% RSLogix 500 project PROC1.RSS, saved by version 8.30.00.16 %
PROJECT "UNTITLED"    % processor: Bul.1763 MicroLogix 1100 Series B %

PROGRAM FILES
  LAD 2 "MAIN"  5 rungs
  LAD 3 "ALARMS"  1 rungs
  LAD 4 "DIGITAL IO"  9 rungs
  LAD 5 "CONTROLS"  1 rungs
  LAD 6 "ANALOG IO"  8 rungs

DATA FILES
  O0 OUTPUT  9 elements
  I1 INPUT  19 elements
  S2 STATUS  66 elements
  B3 BINARY  1 elements
  T4 TIMER  1 elements
  C5 COUNTER  1 elements
  R6 CONTROL  1 elements
  N7 INTEGER  1 elements
  F8 FLOAT  1 elements

LADDER 2 "MAIN"
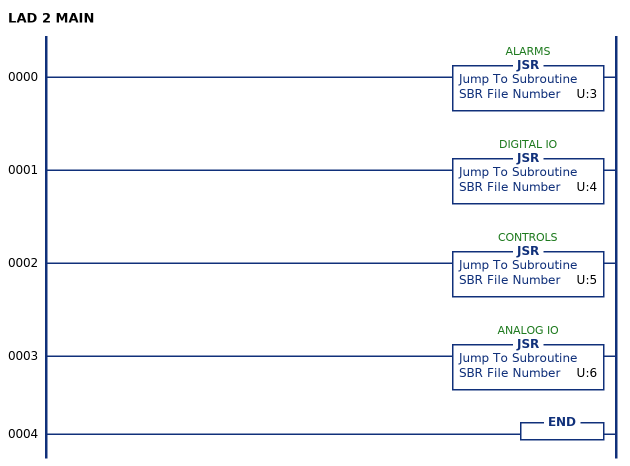
% Rung: 0 %  % edit flag set %
SOR JSR U:3 EOR
%   U:3  "ALARMS" %
% Rung: 1 %
SOR JSR U:4 EOR
%   U:4  "DIGITAL IO" %
% Rung: 2 %  % edit flag set %
SOR JSR U:5 EOR
%   U:5  "CONTROLS" %
% Rung: 3 %  % edit flag set %
SOR JSR U:6 EOR
%   U:6  "ANALOG IO" %
% Rung: 4 %
SOR END EOR

LADDER 4 "DIGITAL IO"
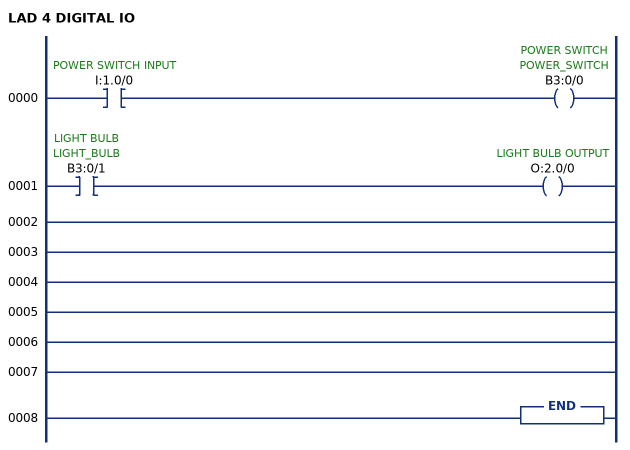
% Rung: 0 %  % edit flag set %
SOR XIC I:1.0/0 OTE B3:0/0 EOR
%   I:1.0/0  "POWER SWITCH INPUT" %
%   B3:0/0  POWER_SWITCH  "POWER SWITCH" %
% Rung: 1 %  % edit flag set %
SOR XIC B3:0/1 OTE O:2.0/0 EOR
%   B3:0/1  LIGHT_BULB  "LIGHT BULB" %
%   O:2.0/0  "LIGHT BULB OUTPUT" %
% Rung: 2 %  % edit flag set %
SOR EOR
% Rung: 3 %  % edit flag set %
SOR EOR
% Rung: 4 %  % edit flag set %
SOR EOR
% Rung: 5 %  % edit flag set %
SOR EOR
% Rung: 6 %  % edit flag set %
SOR EOR
% Rung: 7 %  % edit flag set %
SOR EOR
% Rung: 8 %
SOR END EOR

LADDER 6 "ANALOG IO"
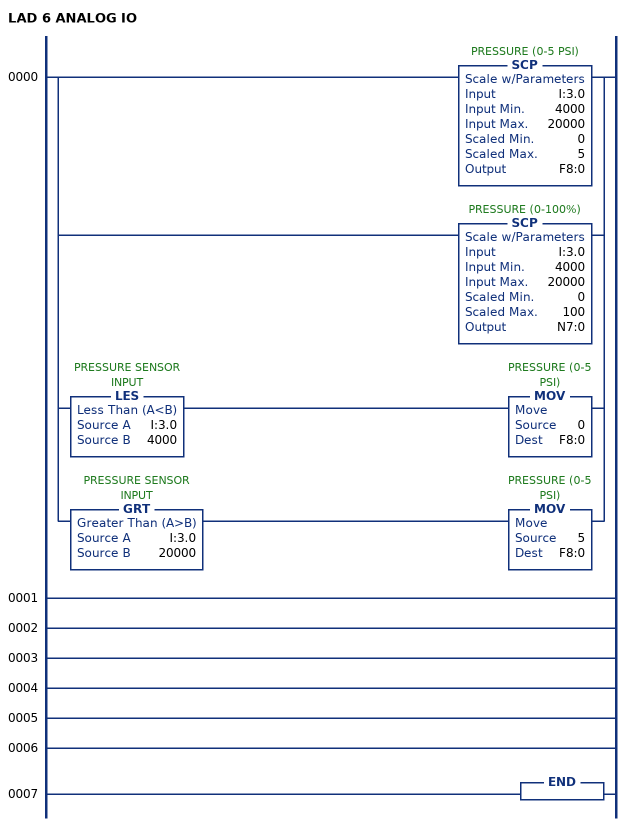
% Rung: 0 %  % edit flag set %
SOR BST SCP I:3.0 4000 20000 0 5 F8:0 NXB SCP I:3.0 4000 20000 0 100 N7:0 NXB LES I:3.0 4000 MOV 0 F8:0 NXB GRT I:3.0 20000 MOV 5 F8:0 BND EOR
%   I:3.0  "PRESSURE SENSOR INPUT" %
%   F8:0  "PRESSURE (0-5 PSI)" %
%   N7:0  "PRESSURE (0-100%)" %
% Rung: 1 %  % edit flag set %
SOR EOR
% Rung: 2 %  % edit flag set %
SOR EOR
% Rung: 3 %  % edit flag set %
SOR EOR
% Rung: 4 %  % edit flag set %
SOR EOR
% Rung: 5 %  % edit flag set %
SOR EOR
% Rung: 6 %  % edit flag set %
SOR EOR
% Rung: 7 %
SOR END EOR

OTHER DOCUMENTED ADDRESSES
  B3:0  TEST_INOUT
  TEST_INPUT  "B3:0"
